PROGRAM Stn055_10_StorageLnSwPrestopGrn
VAR
	{attribute 'TcLinkToOSO' := '.iPuckPresent := <0,1,1>TIIB[N62S00 (AL1332)]^N62S01 (AL2341)^TxPDO^input byte 0;
		.oStopLower := <0,1,1>TIIB[N62S00 (AL1332)]^N62S02 (EX260)^RxPDO^output byte 0'}
	fbConvStop: FB_ConvStop;
END_VAR

//  This code instantiates a component that is implimented as a common function block
//    Note that I/O is linked directly to I/O variables inside the named instance

gStn055_10_StorageLnSwPrestopGrn.ConvRunning := gStn055_16_StorageLnSw.BoschInfeedConvRunning;

fbConvStop(
	pStn := ADR(gStn055),
	pCmp := ADR(gStn055_10_StorageLnSwPrestopGrn),
	pUpstreamStop := 0,
	pStateTraceBuffer := ADR(gStn055_StateTraceBuffer),
	pStateTraceFifo := ADR(gStn055_StateTraceFifo),
	pStats := ADR(gStn055_02_Stats));

END_PROGRAM

(* stored: Version 1.1.0.1, ProductVersion 3.1.4024.6
   POU Stn055_10_StorageLnSwPrestopGrn: Id {dc7f5917-7452-4662-b646-ffb1b5a1e003}, SpecialFunc None *)
